// TIA Portal V20 export
// export: Created 2026-10-01T21:41:12.6332041Z, ExportSetting WithDefaults, DisplayName Totally Integrated Automation Portal, DisplayVersion V20, DisplayName TIA Portal Openness, DisplayVersion V20, DisplayName TIA Portal Version Control Interface, DisplayVersion V20, DisplayName SINAMICS Startdrive Advanced, DisplayVersion V20, DisplayName SINAMICS Startdrive G130, G150, S120, S150, SINAMICS MV, G220, S200, S210, DisplayVersion V20, DisplayName SINAMICS Startdrive G110M, G120, G120C, G120D, G120P, G115D, DisplayVersion V20, DisplayName STEP 7 Professional, DisplayVersion V20, DisplayName STEP 7 Safety, DisplayVersion V20, DisplayName WinCC Basic/Comfort/Advanced, DisplayVersion V20, DisplayName WinCC Unified, DisplayVersion V20
FUNCTION_BLOCK "ZZ_LadTest_Elems"   // FB20, LAD
{ S7_Optimized_Access := 'TRUE' }
VERSION : 0.1
// stored: AutoNumber true, IsIECCheckEnabled false, IsRetainMemResEnabled false, MemoryReserve 100, SetENOAutomatically false, UDAEnableTagReadback false
   VAR_INPUT
      Start : Bool;
      Level : Int;
   END_VAR
   VAR_OUTPUT
      Run : Bool;
      Off : Bool;
      Pulse : Bool;
      Three : Bool;
   END_VAR
   VAR
      Toff : TOF_TIME;
      Tp : TP_TIME;
      Edge1 : Bool;
      Edge2 : Bool;
      "Counter" : Int;
   END_VAR
   VAR_TEMP   // added for the SCL form of the ladder/FBD networks
      _w1 : Bool;
   END_VAR
BEGIN

REGION Network 1
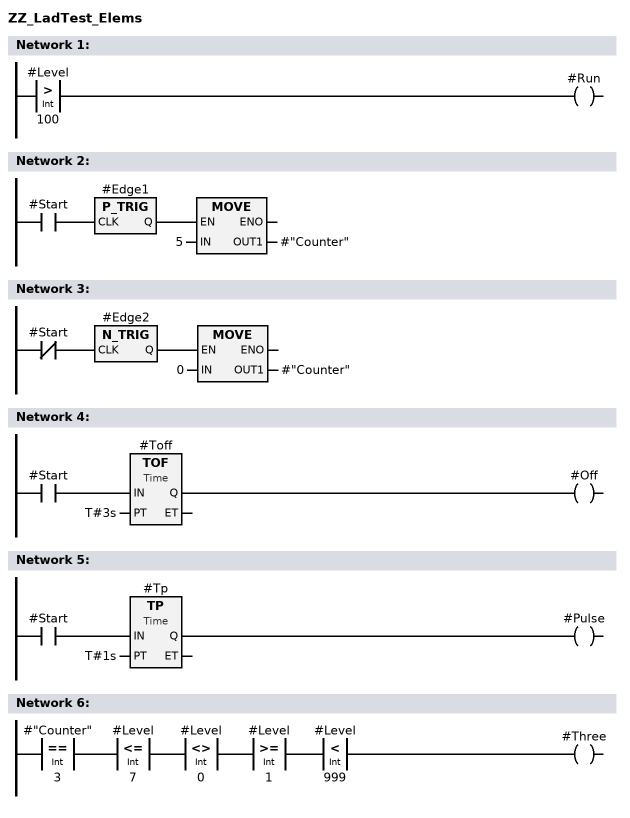
   RUNG wire#powerrail
      { S7_Templates := "SrcType := Int" } GT_Contact(in1 := #Level, in2 := 100)
      Coil( #Run )
   END_RUNG
   // the same network as SCL:
   #Run := #Level > 100;
END_REGION

REGION Network 2
   RUNG wire#powerrail
      Contact( #Start )
      P_Trig( #Edge1 )
      Move(in := 5, out1 => #"Counter")
   END_RUNG
   // the same network as SCL:
   #_w1 := #Start AND NOT #Edge1;   // rising edge
   #Edge1 := #Start;
   IF #_w1 THEN #"Counter" := 5; END_IF;
END_REGION

REGION Network 3
   RUNG wire#powerrail
      I_Contact( #Start )
      N_Trig( #Edge2 )
      Move(in := 0, out1 => #"Counter")
   END_RUNG
   // the same network as SCL:
   #_w1 := NOT (NOT #Start) AND #Edge2;   // falling edge
   #Edge2 := NOT #Start;
   IF #_w1 THEN #"Counter" := 0; END_IF;
END_REGION

REGION Network 4
   RUNG wire#powerrail
      Contact( #Start )
      { S7_Templates := "time_type := Time" } #Toff.TOF(pt := T#3s, et =>)
      Coil( #Off )
   END_RUNG
   // the same network as SCL:
   #Toff(IN := #Start, PT := T#3s);   // TOF
   #Off := #Toff.Q;
END_REGION

REGION Network 5
   RUNG wire#powerrail
      Contact( #Start )
      { S7_Templates := "time_type := Time" } #Tp.TP(pt := T#1s, et =>)
      Coil( #Pulse )
   END_RUNG
   // the same network as SCL:
   #Tp(IN := #Start, PT := T#1s);   // TP
   #Pulse := #Tp.Q;
END_REGION

REGION Network 6
   RUNG wire#powerrail
      { S7_Templates := "SrcType := Int" } EQ_Contact(in1 := #"Counter", in2 := 3)
      { S7_Templates := "SrcType := Int" } LE_Contact(in1 := #Level, in2 := 7)
      { S7_Templates := "SrcType := Int" } NE_Contact(in1 := #Level, in2 := 0)
      { S7_Templates := "SrcType := Int" } GE_Contact(in1 := #Level, in2 := 1)
      { S7_Templates := "SrcType := Int" } LT_Contact(in1 := #Level, in2 := 999)
      Coil( #Three )
   END_RUNG
   // the same network as SCL:
   #Three := (#"Counter" = 3) AND (#Level <= 7) AND (#Level <> 0) AND (#Level >= 1) AND (#Level < 999);
END_REGION
END_FUNCTION_BLOCK
